TYPE OperatingMode :
STRUCT
	ManuelIsActive	:	BOOL;
	AutomaticIsActive	:	BOOL;
	EStop			:	ActionState;
	Fault			:	FaultWarningState;
	Warning			:	FaultWarningState;
	AutomaticStart	:	ActionState;
	AutomaticStop	:	ActionState;
	Reset	:	ActionState;
	Quit	:	ActionState;
	AutomaticHome	:	OperatingModeHomeing;
END_STRUCT
END_TYPE

(* stored: Version 1.1.0.1
   DUT OperatingMode: Id {73b6fc16-f060-4293-9ee5-c29acd1058c2} *)
